TYPE ST_TechnosoftMotionError :
STRUCT
    bEtherCATCommunicationError: BIT; //EtherCAT communication error, bit 0
    bShortCircuit: BIT; //Short circuit, bit 1
    bInvalidSetupData: BIT; //Invalid setup data, bit2
    bControlError: BIT; //Position or speed error, bit3
    bCommunicationError: BIT; //Communication error, bit 4
    bFeedbackError: BIT; //Feedback error, bit 5
    bPositiveLimitSwitchActive: BIT; //Positive limit active, bit 6
    bNegativeLimitSwitchActive: BIT; //Negative limit active, bit 7
    bOverCurrent: BIT; //Over current, bit 8
    bI2TProtection: BIT; //I2T protection active, bit 9
    bMotorOverTemperature: BIT; //Motor over temperature, bit 10
    bDriveOverTemperature: BIT; //Drive over temperature, bit 11
    bOverVoltage: BIT; //Over voltage, bit 12
    bUnderVoltage: BIT; //Under voltage, bit 13
    bCommandError: BIT; //Command error, bit 14
    bSTOActive: BIT; //Enabled or STO disabled, bit 15
END_STRUCT
END_TYPE

(* stored: Version 1.1.0.1
   DUT ST_TechnosoftMotionError: Id {90598514-2df2-078a-0a1a-d8b0c6c1a1f5} *)
